{attribute 'qualified_only'}
{attribute 'strict'}
TYPE ePumpState :
(
	Off := 0,
	Starting := 1,
	Running	:= 2,
	Stopping := 3
);
END_TYPE

(* stored: Version 1.1.0.1, ProductVersion 3.1.4024.12
   DUT ePumpState: Id {99455111-0b92-4620-90ef-cfb6cb9aff3a} *)
